PROGRAM MAIN_KOLMI
VAR
END_VAR

END_PROGRAM

(* stored: Version 1.1.0.1, ProductVersion 3.1.4024.6
   POU MAIN_KOLMI: Id {48d5b021-12c4-493c-a120-e4027bfa7c90}, SpecialFunc None *)
